// TIA Portal project "functon block" (V15)

(* hardware
DEVICE "S7-1200 station_1"  S7-1200 Station
   slot 0: "Rack_0"  S7-1200 Rack  Rack  V1.0
   slot 1: "PLC_1"  CPU 1214C DC/DC/DC  6ES7 214-1AG40-0XB0  V4.2
   slot 2: "AI 4x13BIT/AQ 2x14BIT_1"  6ES7 234-4HE32-0XB0  V2.0
   slot 101: "CM 1241 (RS422/485)_1"  6ES7 241-1CH32-0XB0  V2.2
*)

// ===== PLC "PLC_1"  CPU 1214C DC/DC/DC =====

VAR_GLOBAL   // PLC tag table "Default tag table"
   "val1" AT %IW0 : Int;
   "val2" AT %IW2 : Int;
   "val3" AT %MW0 : Int;
   "in1" AT %MW2 : Int;
   "in2" AT %MW4 : Int;
   "switch" AT %M6.0 : Bool;
END_VAR

FUNCTION "adder" : Void   // FC1, LAD
{ S7_Optimized_Access := 'TRUE' }
VERSION : 0.1
   VAR_INPUT
      loc1 : Int;
      loc2 : Int;
   END_VAR
BEGIN

REGION Network 1
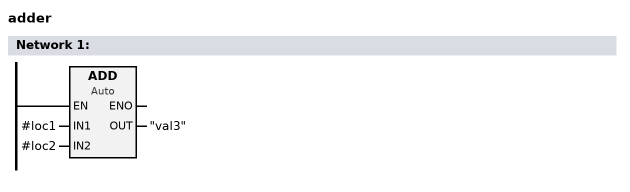
   RUNG wire#powerrail
      Add(in1 := #loc1, in2 := #loc2, out => "val3")
   END_RUNG
   // the same network as SCL:
   "val3" := #loc1 + #loc2;
END_REGION
END_FUNCTION

ORGANIZATION_BLOCK "Main"   // OB1, LAD, ProgramCycle
TITLE = "Main Program Sweep (Cycle)"
{ S7_Optimized_Access := 'TRUE' }
VERSION : 0.1
   VAR_INPUT
      Initial_Call : Bool;   // Initial call of this OB
      Remanence : Bool;   // =True, if remanent data are available
   END_VAR
   VAR_TEMP
      out : Int;
   END_VAR
BEGIN

REGION Network 1
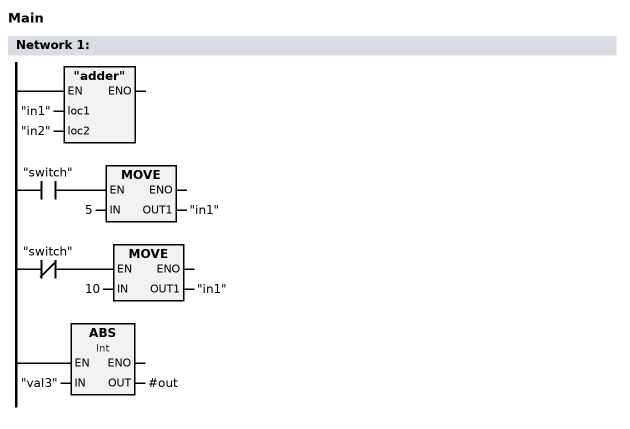
   RUNG wire#powerrail
      "adder"(loc1 := "in1", loc2 := "in2")
   END_RUNG
   RUNG wire#powerrail
      Contact( "switch" )
      Move(in := 5, out1 => "in1")
   END_RUNG
   RUNG wire#powerrail
      I_Contact( "switch" )
      Move(in := 10, out1 => "in1")
   END_RUNG
   RUNG wire#powerrail
      { S7_Templates := "SrcType := Int" } Abs(in := "val3", out => #out)
   END_RUNG
   // the same network as SCL:
   "adder"(loc1 := "in1", loc2 := "in2");
   IF "switch" THEN "in1" := 5; END_IF;
   IF NOT "switch" THEN "in1" := 10; END_IF;
   #out := ABS("val3");
END_REGION
END_ORGANIZATION_BLOCK